PROGRAM MAIN_TEST
VAR
END_VAR

END_PROGRAM

(* stored: Version 1.1.0.1, ProductVersion 3.1.4022.18
   POU MAIN_TEST: Id {e0fe771e-7548-4546-bb6c-2059f20a9739}, SpecialFunc None *)
